PROGRAM MAIN
VAR
	fbSequenceManager	: FB_SequenceManager;
	nTest				: INT;
END_VAR

IF (nTest = 1) THEN
	fbSequenceManager.Sort(E_SortedOrder.Id, E_SortedDirection.Ascending);
	nTest := 0;
ELSIF (nTest = 2) THEN
	fbSequenceManager.Sort(E_SortedOrder.Value, E_SortedDirection.Ascending);
	nTest := 0;
ELSIF (nTest = 3) THEN
	fbSequenceManager.Sort(E_SortedOrder.Duration, E_SortedDirection.Ascending);
	nTest := 0;
ELSIF (nTest = 4) THEN
	fbSequenceManager.Sort(E_SortedOrder.Id, E_SortedDirection.Descending);
	nTest := 0;
ELSIF (nTest = 5) THEN
	fbSequenceManager.Sort(E_SortedOrder.Value, E_SortedDirection.Descending);
	nTest := 0;
ELSIF (nTest = 6) THEN
	fbSequenceManager.Sort(E_SortedOrder.Duration, E_SortedDirection.Descending);
	nTest := 0;
END_IF

END_PROGRAM

(* stored: Version 1.1.0.1, ProductVersion 3.1.4024.12
   POU MAIN: Id {97b18291-6e7e-4445-af9e-8a6ad63835f0}, SpecialFunc None *)
